TYPE ASCF_CC_OPCUACS_WriterStatus :
STRUCT
	State		: WORD		:= 16#0;
	Error		: BOOL		:= FALSE;
	Status		: DWORD		:= 16#0;
	Cycle		: TIME		:= T#0MS;
END_STRUCT
END_TYPE

(* stored: Version 1.1.0.1, ProductVersion 3.1.4026.4
   DUT ASCF_CC_OPCUACS_WriterStatus: Id {db1f49b9-3e03-43fb-8512-9a7f1394e91e} *)
